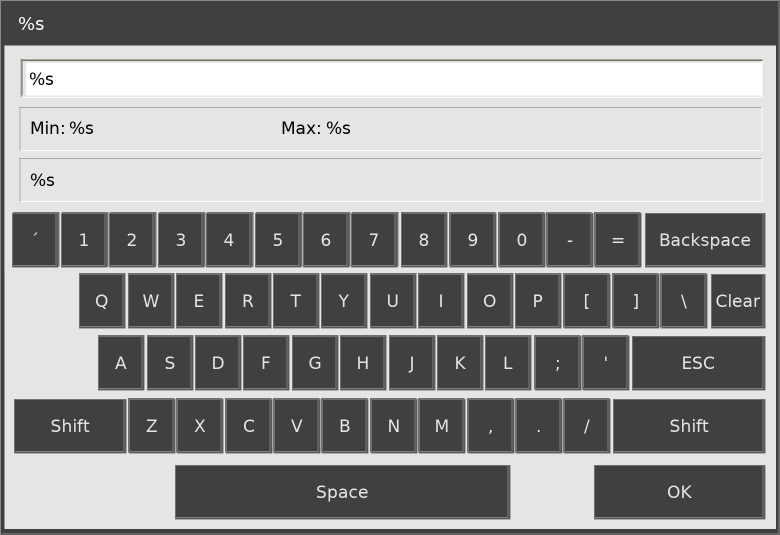
VISUALIZATION Keypad  // 780x535
VAR_INPUT
	stVariableValue 						: STRING;
	stMin 									: STRING;
	stMax 									: STRING;
	stTitle 								: STRING;
	flags 									: DWORD;
END_VAR
VAR
	bInit 									: BOOL;
	bShift 									: BOOL;
	stMessage 								: STRING;
	stOutputValue 							: STRING;
END_VAR
    Rectangle (5,201 772x70)
    Rectangle (3,271 775x62)
    Rectangle (3,333 775x63)
    Rectangle (3,396 775x62)
    Rectangle (3,455 775x75)
    Button (594,465 171x54), "OK"
        OnMouseDown: CloseDialog Dialog=Keypad, Result=OK, NumpadKeypad=True, NumpadKeypadSet=True
    Button (632,336 133x54), "ESC"
        OnMouseDown: CloseDialog Dialog=Keypad, Result=Cancel, NumpadKeypad=True, NumpadKeypadSet=True
    Button (711,274 54x54), "Clear"
        OnMouseDown: execute { stVariableValue := ''; stOutputValue := ''; }
    Button (645,213 120x54), "Backspace"
        OnMouseDown: execute { VisuDlg_CheckedBack(stOutputValue, stVariableValue, bInit); }
    Button (613,399 152x54), "Shift"
        OnMouseDown: toggle bShift
    Button (175,465 335x54), "Space"
        OnMouseDown: execute { VisuDlg_CheckedAppend(stOutputValue, stVariableValue, bInit, (flags AND VisuElems.Visu_InputFlags.Password) = 1, ' '); }
    Button (660,273 46x54), "|", invisible if: NOT bShift
        OnMouseDown: execute { VisuDlg_CheckedAppend(stOutputValue, stVariableValue, bInit, (flags AND VisuElems.Visu_InputFlags.Password) = 1, '|'); }
    Button (467,398 46x54), "<", invisible if: NOT bShift
        OnMouseDown: execute { VisuDlg_CheckedAppend(stOutputValue, stVariableValue, bInit, (flags AND VisuElems.Visu_InputFlags.Password) = 1, '<'); }
    Button (515,398 46x54), ">", invisible if: NOT bShift
        OnMouseDown: execute { VisuDlg_CheckedAppend(stOutputValue, stVariableValue, bInit, (flags AND VisuElems.Visu_InputFlags.Password) = 1, '>'); }
    Button (321,273 46x54), "y", invisible if: NOT bShift
        OnMouseDown: execute { VisuDlg_CheckedAppend(stOutputValue, stVariableValue, bInit, (flags AND VisuElems.Visu_InputFlags.Password) = 1, 'y'); }
    Button (321,274 46x54), "Y", invisible if: bShift
        OnMouseDown: execute { VisuDlg_CheckedAppend(stOutputValue, stVariableValue, bInit, (flags AND VisuElems.Visu_InputFlags.Password) = 1, 'Y'); }
    Button (176,398 46x54), "x", invisible if: NOT bShift
        OnMouseDown: execute { VisuDlg_CheckedAppend(stOutputValue, stVariableValue, bInit, (flags AND VisuElems.Visu_InputFlags.Password) = 1, 'x'); }
    Button (177,399 46x54), "X", invisible if: bShift
        OnMouseDown: execute { VisuDlg_CheckedAppend(stOutputValue, stVariableValue, bInit, (flags AND VisuElems.Visu_InputFlags.Password) = 1, 'X'); }
    Button (225,398 46x54), "c", invisible if: NOT bShift
        OnMouseDown: execute { VisuDlg_CheckedAppend(stOutputValue, stVariableValue, bInit, (flags AND VisuElems.Visu_InputFlags.Password) = 1, 'c'); }
    Button (226,399 46x54), "C", invisible if: bShift
        OnMouseDown: execute { VisuDlg_CheckedAppend(stOutputValue, stVariableValue, bInit, (flags AND VisuElems.Visu_InputFlags.Password) = 1, 'C'); }
    Button (273,398 46x54), "v", invisible if: NOT bShift
        OnMouseDown: execute { VisuDlg_CheckedAppend(stOutputValue, stVariableValue, bInit, (flags AND VisuElems.Visu_InputFlags.Password) = 1, 'v'); }
    Button (274,399 46x54), "V", invisible if: bShift
        OnMouseDown: execute { VisuDlg_CheckedAppend(stOutputValue, stVariableValue, bInit, (flags AND VisuElems.Visu_InputFlags.Password) = 1, 'V'); }
    Button (321,398 46x54), "b", invisible if: NOT bShift
        OnMouseDown: execute { VisuDlg_CheckedAppend(stOutputValue, stVariableValue, bInit, (flags AND VisuElems.Visu_InputFlags.Password) = 1, 'b'); }
    Button (322,399 46x54), "B", invisible if: bShift
        OnMouseDown: execute { VisuDlg_CheckedAppend(stOutputValue, stVariableValue, bInit, (flags AND VisuElems.Visu_InputFlags.Password) = 1, 'B'); }
    Button (370,398 46x54), "n", invisible if: NOT bShift
        OnMouseDown: execute { VisuDlg_CheckedAppend(stOutputValue, stVariableValue, bInit, (flags AND VisuElems.Visu_InputFlags.Password) = 1, 'n'); }
    Button (371,399 46x54), "N", invisible if: bShift
        OnMouseDown: execute { VisuDlg_CheckedAppend(stOutputValue, stVariableValue, bInit, (flags AND VisuElems.Visu_InputFlags.Password) = 1, 'N'); }
    Button (418,398 46x54), "m", invisible if: NOT bShift
        OnMouseDown: execute { VisuDlg_CheckedAppend(stOutputValue, stVariableValue, bInit, (flags AND VisuElems.Visu_InputFlags.Password) = 1, 'm'); }
    Button (419,399 46x54), "M", invisible if: bShift
        OnMouseDown: execute { VisuDlg_CheckedAppend(stOutputValue, stVariableValue, bInit, (flags AND VisuElems.Visu_InputFlags.Password) = 1, 'M'); }
    Button (534,335 46x54), ":", invisible if: NOT bShift
        OnMouseDown: execute { VisuDlg_CheckedAppend(stOutputValue, stVariableValue, bInit, (flags AND VisuElems.Visu_InputFlags.Password) = 1, ':'); }
    Button (546,212 45x54), "_", invisible if: NOT bShift
        OnMouseDown: execute { VisuDlg_CheckedAppend(stOutputValue, stVariableValue, bInit, (flags AND VisuElems.Visu_InputFlags.Password) = 1, '_'); }
    Button (98,335 46x54), "a", invisible if: NOT bShift
        OnMouseDown: execute { VisuDlg_CheckedAppend(stOutputValue, stVariableValue, bInit, (flags AND VisuElems.Visu_InputFlags.Password) = 1, 'a'); }
    Button (98,336 46x54), "A", invisible if: bShift
        OnMouseDown: execute { VisuDlg_CheckedAppend(stOutputValue, stVariableValue, bInit, (flags AND VisuElems.Visu_InputFlags.Password) = 1, 'A'); }
    Button (147,335 46x54), "s", invisible if: NOT bShift
        OnMouseDown: execute { VisuDlg_CheckedAppend(stOutputValue, stVariableValue, bInit, (flags AND VisuElems.Visu_InputFlags.Password) = 1, 's'); }
    Button (147,336 46x54), "S", invisible if: bShift
        OnMouseDown: execute { VisuDlg_CheckedAppend(stOutputValue, stVariableValue, bInit, (flags AND VisuElems.Visu_InputFlags.Password) = 1, 'S'); }
    Button (195,335 46x54), "d", invisible if: NOT bShift
        OnMouseDown: execute { VisuDlg_CheckedAppend(stOutputValue, stVariableValue, bInit, (flags AND VisuElems.Visu_InputFlags.Password) = 1, 'd'); }
    Button (195,336 46x54), "D", invisible if: bShift
        OnMouseDown: execute { VisuDlg_CheckedAppend(stOutputValue, stVariableValue, bInit, (flags AND VisuElems.Visu_InputFlags.Password) = 1, 'D'); }
    Button (243,335 46x54), "f", invisible if: NOT bShift
        OnMouseDown: execute { VisuDlg_CheckedAppend(stOutputValue, stVariableValue, bInit, (flags AND VisuElems.Visu_InputFlags.Password) = 1, 'f'); }
    Button (243,336 46x54), "F", invisible if: bShift
        OnMouseDown: execute { VisuDlg_CheckedAppend(stOutputValue, stVariableValue, bInit, (flags AND VisuElems.Visu_InputFlags.Password) = 1, 'F'); }
    Button (292,335 46x54), "g", invisible if: NOT bShift
        OnMouseDown: execute { VisuDlg_CheckedAppend(stOutputValue, stVariableValue, bInit, (flags AND VisuElems.Visu_InputFlags.Password) = 1, 'g'); }
    Button (292,336 46x54), "G", invisible if: bShift
        OnMouseDown: execute { VisuDlg_CheckedAppend(stOutputValue, stVariableValue, bInit, (flags AND VisuElems.Visu_InputFlags.Password) = 1, 'G'); }
    Button (340,335 46x54), "h", invisible if: NOT bShift
        OnMouseDown: execute { VisuDlg_CheckedAppend(stOutputValue, stVariableValue, bInit, (flags AND VisuElems.Visu_InputFlags.Password) = 1, 'h'); }
    Button (340,336 46x54), "H", invisible if: bShift
        OnMouseDown: execute { VisuDlg_CheckedAppend(stOutputValue, stVariableValue, bInit, (flags AND VisuElems.Visu_InputFlags.Password) = 1, 'H'); }
    Button (389,335 46x54), "j", invisible if: NOT bShift
        OnMouseDown: execute { VisuDlg_CheckedAppend(stOutputValue, stVariableValue, bInit, (flags AND VisuElems.Visu_InputFlags.Password) = 1, 'j'); }
    Button (389,336 46x54), "J", invisible if: bShift
        OnMouseDown: execute { VisuDlg_CheckedAppend(stOutputValue, stVariableValue, bInit, (flags AND VisuElems.Visu_InputFlags.Password) = 1, 'J'); }
    Button (437,335 46x54), "k", invisible if: NOT bShift
        OnMouseDown: execute { VisuDlg_CheckedAppend(stOutputValue, stVariableValue, bInit, (flags AND VisuElems.Visu_InputFlags.Password) = 1, 'k'); }
    Button (437,336 46x54), "K", invisible if: bShift
        OnMouseDown: execute { VisuDlg_CheckedAppend(stOutputValue, stVariableValue, bInit, (flags AND VisuElems.Visu_InputFlags.Password) = 1, 'K'); }
    Button (485,335 46x54), "l", invisible if: NOT bShift
        OnMouseDown: execute { VisuDlg_CheckedAppend(stOutputValue, stVariableValue, bInit, (flags AND VisuElems.Visu_InputFlags.Password) = 1, 'l'); }
    Button (485,336 46x54), "L", invisible if: bShift
        OnMouseDown: execute { VisuDlg_CheckedAppend(stOutputValue, stVariableValue, bInit, (flags AND VisuElems.Visu_InputFlags.Password) = 1, 'L'); }
    Button (159,212 46x54), "#", invisible if: NOT bShift
        OnMouseDown: execute { VisuDlg_CheckedAppend(stOutputValue, stVariableValue, bInit, (flags AND VisuElems.Visu_InputFlags.Password) = 1, '#'); }
    Button (110,212 46x54), "@", invisible if: NOT bShift
        OnMouseDown: execute { VisuDlg_CheckedAppend(stOutputValue, stVariableValue, bInit, (flags AND VisuElems.Visu_InputFlags.Password) = 1, '@'); }
    Button (79,273 46x54), "q", invisible if: NOT bShift
        OnMouseDown: execute { VisuDlg_CheckedAppend(stOutputValue, stVariableValue, bInit, (flags AND VisuElems.Visu_InputFlags.Password) = 1, 'q'); }
    Button (79,274 46x54), "Q", invisible if: bShift
        OnMouseDown: execute { VisuDlg_CheckedAppend(stOutputValue, stVariableValue, bInit, (flags AND VisuElems.Visu_InputFlags.Password) = 1, 'Q'); }
    Button (128,273 46x54), "w", invisible if: NOT bShift
        OnMouseDown: execute { VisuDlg_CheckedAppend(stOutputValue, stVariableValue, bInit, (flags AND VisuElems.Visu_InputFlags.Password) = 1, 'w'); }
    Button (128,274 46x54), "W", invisible if: bShift
        OnMouseDown: execute { VisuDlg_CheckedAppend(stOutputValue, stVariableValue, bInit, (flags AND VisuElems.Visu_InputFlags.Password) = 1, 'W'); }
    Button (176,273 46x54), "e", invisible if: NOT bShift
        OnMouseDown: execute { VisuDlg_CheckedAppend(stOutputValue, stVariableValue, bInit, (flags AND VisuElems.Visu_InputFlags.Password) = 1, 'e'); }
    Button (176,274 46x54), "E", invisible if: bShift
        OnMouseDown: execute { VisuDlg_CheckedAppend(stOutputValue, stVariableValue, bInit, (flags AND VisuElems.Visu_InputFlags.Password) = 1, 'E'); }
    Button (225,273 46x54), "r", invisible if: NOT bShift
        OnMouseDown: execute { VisuDlg_CheckedAppend(stOutputValue, stVariableValue, bInit, (flags AND VisuElems.Visu_InputFlags.Password) = 1, 'r'); }
    Button (225,274 46x54), "R", invisible if: bShift
        OnMouseDown: execute { VisuDlg_CheckedAppend(stOutputValue, stVariableValue, bInit, (flags AND VisuElems.Visu_InputFlags.Password) = 1, 'R'); }
    Button (273,273 46x54), "t", invisible if: NOT bShift
        OnMouseDown: execute { VisuDlg_CheckedAppend(stOutputValue, stVariableValue, bInit, (flags AND VisuElems.Visu_InputFlags.Password) = 1, 't'); }
    Button (273,274 46x54), "T", invisible if: bShift
        OnMouseDown: execute { VisuDlg_CheckedAppend(stOutputValue, stVariableValue, bInit, (flags AND VisuElems.Visu_InputFlags.Password) = 1, 'T'); }
    Button (128,398 46x54), "z", invisible if: NOT bShift
        OnMouseDown: execute { VisuDlg_CheckedAppend(stOutputValue, stVariableValue, bInit, (flags AND VisuElems.Visu_InputFlags.Password) = 1, 'z'); }
    Button (129,399 46x54), "Z", invisible if: bShift
        OnMouseDown: execute { VisuDlg_CheckedAppend(stOutputValue, stVariableValue, bInit, (flags AND VisuElems.Visu_InputFlags.Password) = 1, 'Z'); }
    Button (370,273 46x54), "u", invisible if: NOT bShift
        OnMouseDown: execute { VisuDlg_CheckedAppend(stOutputValue, stVariableValue, bInit, (flags AND VisuElems.Visu_InputFlags.Password) = 1, 'u'); }
    Button (370,274 46x54), "U", invisible if: bShift
        OnMouseDown: execute { VisuDlg_CheckedAppend(stOutputValue, stVariableValue, bInit, (flags AND VisuElems.Visu_InputFlags.Password) = 1, 'U'); }
    Button (418,273 46x54), "i", invisible if: NOT bShift
        OnMouseDown: execute { VisuDlg_CheckedAppend(stOutputValue, stVariableValue, bInit, (flags AND VisuElems.Visu_InputFlags.Password) = 1, 'i'); }
    Button (418,274 46x54), "I", invisible if: bShift
        OnMouseDown: execute { VisuDlg_CheckedAppend(stOutputValue, stVariableValue, bInit, (flags AND VisuElems.Visu_InputFlags.Password) = 1, 'I'); }
    Button (467,273 46x54), "o", invisible if: NOT bShift
        OnMouseDown: execute { VisuDlg_CheckedAppend(stOutputValue, stVariableValue, bInit, (flags AND VisuElems.Visu_InputFlags.Password) = 1, 'o'); }
    Button (467,274 46x54), "O", invisible if: bShift
        OnMouseDown: execute { VisuDlg_CheckedAppend(stOutputValue, stVariableValue, bInit, (flags AND VisuElems.Visu_InputFlags.Password) = 1, 'O'); }
    Button (515,273 46x54), "p", invisible if: NOT bShift
        OnMouseDown: execute { VisuDlg_CheckedAppend(stOutputValue, stVariableValue, bInit, (flags AND VisuElems.Visu_InputFlags.Password) = 1, 'p'); }
    Button (515,274 46x54), "P", invisible if: bShift
        OnMouseDown: execute { VisuDlg_CheckedAppend(stOutputValue, stVariableValue, bInit, (flags AND VisuElems.Visu_InputFlags.Password) = 1, 'P'); }
    Button (594,212 46x54), "+", invisible if: NOT bShift
        OnMouseDown: execute { VisuDlg_CheckedAppend(stOutputValue, stVariableValue, bInit, (flags AND VisuElems.Visu_InputFlags.Password) = 1, '+'); }
    Button (401,212 46x54), "*", invisible if: NOT bShift
        OnMouseDown: execute { VisuDlg_CheckedAppend(stOutputValue, stVariableValue, bInit, (flags AND VisuElems.Visu_InputFlags.Password) = 1, '*'); }
    Button (13,212 46x54), "~", invisible if: NOT bShift
        OnMouseDown: execute { VisuDlg_CheckedAppend(stOutputValue, stVariableValue, bInit, (flags AND VisuElems.Visu_InputFlags.Password) = 1, '~'); }
    Button (304,212 46x54), "^", invisible if: NOT bShift
        OnMouseDown: execute { VisuDlg_CheckedAppend(stOutputValue, stVariableValue, bInit, (flags AND VisuElems.Visu_InputFlags.Password) = 1, '^'); }
    Button (62,212 46x54), "!", invisible if: NOT bShift
        OnMouseDown: execute { VisuDlg_CheckedAppend(stOutputValue, stVariableValue, bInit, (flags AND VisuElems.Visu_InputFlags.Password) = 1, '!'); }
    Button (582,335 46x54), """, invisible if: NOT bShift
        OnMouseDown: execute { VisuDlg_CheckedAppend(stOutputValue, stVariableValue, bInit, (flags AND VisuElems.Visu_InputFlags.Password) = 1, '"'); }
    Button (207,212 46x54), "$", invisible if: NOT bShift
        OnMouseDown: execute { VisuDlg_CheckedAppend(stOutputValue, stVariableValue, bInit, (flags AND VisuElems.Visu_InputFlags.Password) = 1, '$$'); }
    Button (256,212 46x54), "%", invisible if: NOT bShift
        OnMouseDown: execute { VisuDlg_CheckedAppend(stOutputValue, stVariableValue, bInit, (flags AND VisuElems.Visu_InputFlags.Password) = 1, '%'); }
    Button (352,212 46x54), "&", invisible if: NOT bShift
        OnMouseDown: execute { VisuDlg_CheckedAppend(stOutputValue, stVariableValue, bInit, (flags AND VisuElems.Visu_InputFlags.Password) = 1, '&'); }
    Button (449,212 46x54), "(", invisible if: NOT bShift
        OnMouseDown: execute { VisuDlg_CheckedAppend(stOutputValue, stVariableValue, bInit, (flags AND VisuElems.Visu_InputFlags.Password) = 1, '('); }
    Button (498,212 46x54), ")", invisible if: NOT bShift
        OnMouseDown: execute { VisuDlg_CheckedAppend(stOutputValue, stVariableValue, bInit, (flags AND VisuElems.Visu_InputFlags.Password) = 1, ')'); }
    Button (563,398 46x54), "?", invisible if: NOT bShift
        OnMouseDown: execute { VisuDlg_CheckedAppend(stOutputValue, stVariableValue, bInit, (flags AND VisuElems.Visu_InputFlags.Password) = 1, '?'); }
    Rectangle (5,104 773x97)
    Rectangle (27,164 734x32), "%s", text variable: stMessage
    Rectangle (5,42 773x62)
    Rectangle (776,0 4x530)
    Rectangle (0,2 4x527)
    Rectangle (0,529 780x6)
    Polyline (20,201) (20,158) (762,158)
    Polyline (20,150) (20,107) (762,107)
    Polyline (21,97) (21,59) (762,59)
    Polyline (21,201) (762,201) (762,158)
    Polyline (21,150) (762,150) (762,107)
    Polyline (22,97) (762,97) (762,60)
    Rectangle (0,0 779x45)
    Rectangle (15,8 757x32), "%s", text variable: stTitle
    Polyline (22,95) (22,60) (762,60)
    Rectangle (26,63 736x32), "%s", text variable: stOutputValue
    Rectangle (27,112 42x32), "Min:", text variable: stMin, invisible if: LEN(stMin) = 0
    Rectangle (66,112 157x32), "%s", text variable: stMin, invisible if: LEN(stMin) = 0
    Rectangle (278,112 45x32), "Max:", text variable: stMin, invisible if: LEN(stMax) = 0
    Rectangle (323,112 217x32), "%s", text variable: stMax, invisible if: LEN(stMax) = 0
    Button (12,213 46x54), "´", invisible if: bShift
        OnMouseDown: execute { VisuDlg_CheckedAppend(stOutputValue, stVariableValue, bInit, (flags AND VisuElems.Visu_InputFlags.Password) = 1, '´'); }
    Button (61,213 46x54), "1", invisible if: bShift
        OnMouseDown: execute { VisuDlg_CheckedAppend(stOutputValue, stVariableValue, bInit, (flags AND VisuElems.Visu_InputFlags.Password) = 1, '1'); }
    Button (109,213 46x54), "2", invisible if: bShift
        OnMouseDown: execute { VisuDlg_CheckedAppend(stOutputValue, stVariableValue, bInit, (flags AND VisuElems.Visu_InputFlags.Password) = 1, '2'); }
    Button (158,213 46x54), "3", invisible if: bShift
        OnMouseDown: execute { VisuDlg_CheckedAppend(stOutputValue, stVariableValue, bInit, (flags AND VisuElems.Visu_InputFlags.Password) = 1, '3'); }
    Button (206,213 46x54), "4", invisible if: bShift
        OnMouseDown: execute { VisuDlg_CheckedAppend(stOutputValue, stVariableValue, bInit, (flags AND VisuElems.Visu_InputFlags.Password) = 1, '4'); }
    Button (255,213 46x54), "5", invisible if: bShift
        OnMouseDown: execute { VisuDlg_CheckedAppend(stOutputValue, stVariableValue, bInit, (flags AND VisuElems.Visu_InputFlags.Password) = 1, '5'); }
    Button (303,213 46x54), "6", invisible if: bShift
        OnMouseDown: execute { VisuDlg_CheckedAppend(stOutputValue, stVariableValue, bInit, (flags AND VisuElems.Visu_InputFlags.Password) = 1, '6'); }
    Button (351,213 46x54), "7", invisible if: bShift
        OnMouseDown: execute { VisuDlg_CheckedAppend(stOutputValue, stVariableValue, bInit, (flags AND VisuElems.Visu_InputFlags.Password) = 1, '7'); }
    Button (401,213 46x54), "8", invisible if: bShift
        OnMouseDown: execute { VisuDlg_CheckedAppend(stOutputValue, stVariableValue, bInit, (flags AND VisuElems.Visu_InputFlags.Password) = 1, '8'); }
    Button (450,213 46x54), "9", invisible if: bShift
        OnMouseDown: execute { VisuDlg_CheckedAppend(stOutputValue, stVariableValue, bInit, (flags AND VisuElems.Visu_InputFlags.Password) = 1, '9'); }
    Button (499,213 46x54), "0", invisible if: bShift
        OnMouseDown: execute { VisuDlg_CheckedAppend(stOutputValue, stVariableValue, bInit, (flags AND VisuElems.Visu_InputFlags.Password) = 1, '0'); }
    Button (547,213 46x54), "-", invisible if: bShift
        OnMouseDown: execute { VisuDlg_CheckedAppend(stOutputValue, stVariableValue, bInit, (flags AND VisuElems.Visu_InputFlags.Password) = 1, '-'); }
    Button (595,213 46x54), "=", invisible if: bShift
        OnMouseDown: execute { VisuDlg_CheckedAppend(stOutputValue, stVariableValue, bInit, (flags AND VisuElems.Visu_InputFlags.Password) = 1, '='); }
    Button (563,273 46x54), "{", invisible if: NOT bShift
        OnMouseDown: execute { VisuDlg_CheckedAppend(stOutputValue, stVariableValue, bInit, (flags AND VisuElems.Visu_InputFlags.Password) = 1, '{'); }
    Button (564,274 46x54), "[", invisible if: bShift
        OnMouseDown: execute { VisuDlg_CheckedAppend(stOutputValue, stVariableValue, bInit, (flags AND VisuElems.Visu_InputFlags.Password) = 1, '['); }
    Button (612,273 46x54), "}", invisible if: NOT bShift
        OnMouseDown: execute { VisuDlg_CheckedAppend(stOutputValue, stVariableValue, bInit, (flags AND VisuElems.Visu_InputFlags.Password) = 1, '}'); }
    Button (613,274 46x54), "]", invisible if: bShift
        OnMouseDown: execute { VisuDlg_CheckedAppend(stOutputValue, stVariableValue, bInit, (flags AND VisuElems.Visu_InputFlags.Password) = 1, ']'); }
    Button (661,274 46x54), "\", invisible if: bShift
        OnMouseDown: execute { VisuDlg_CheckedAppend(stOutputValue, stVariableValue, bInit, (flags AND VisuElems.Visu_InputFlags.Password) = 1, '\'); }
    Button (535,336 46x54), ";", invisible if: bShift
        OnMouseDown: execute { VisuDlg_CheckedAppend(stOutputValue, stVariableValue, bInit, (flags AND VisuElems.Visu_InputFlags.Password) = 1, ';'); }
    Button (583,336 46x54), "'", invisible if: bShift
        OnMouseDown: execute { VisuDlg_CheckedAppend(stOutputValue, stVariableValue, bInit, (flags AND VisuElems.Visu_InputFlags.Password) = 1, '$''); }
    Button (468,399 46x54), ",", invisible if: bShift
        OnMouseDown: execute { VisuDlg_CheckedAppend(stOutputValue, stVariableValue, bInit, (flags AND VisuElems.Visu_InputFlags.Password) = 1, ','); }
    Button (516,399 46x54), ".", invisible if: bShift
        OnMouseDown: execute { VisuDlg_CheckedAppend(stOutputValue, stVariableValue, bInit, (flags AND VisuElems.Visu_InputFlags.Password) = 1, '.'); }
    Button (564,399 46x54), "/", invisible if: bShift
        OnMouseDown: execute { VisuDlg_CheckedAppend(stOutputValue, stVariableValue, bInit, (flags AND VisuElems.Visu_InputFlags.Password) = 1, '/'); }
    Button (14,399 112x54), "Shift"
        OnMouseDown: toggle bShift
    hotkey HotkeyInput Id=481083523072, Key=KeyDown=True, KeyName=BACKSPACE, ActionToExecute=Action=STSnippet=VisuDlg_CheckedBack(stOutputValue, stVariableValue, bInit);, VisuElemId=-1
    hotkey HotkeyInput Id=481084571648, Key=KeyDown=True, KeyName=DELETE, ActionToExecute=Action=STSnippet=stVariableValue := ''; stOutputValue := '';, VisuElemId=-1
    hotkey HotkeyInput Id=481085620224, Key=KeyDown=True, KeyName=ESCAPE, ActionToExecute=Action=Dialog=Keypad, Result=Cancel, NumpadKeypad=True, NumpadKeypadSet=True, VisuElemId=-1
    hotkey HotkeyInput Id=481086668800, Key=KeyDown=True, KeyName=SPACE, ActionToExecute=Action=STSnippet=VisuDlg_CheckedAppend(stOutputValue, stVariableValue, bInit, (flags AND VisuElems.Visu_InputFlags.Password) = 1, ' ');, VisuElemId=-1
    hotkey HotkeyInput Id=481087717376, Key=Modifiers=1, KeyDown=True, KeyName=SPACE, ActionToExecute=Action=ToggleVariable=bShift, VisuElemId=-1
    hotkey HotkeyInput Id=481088765952, Key=KeyDown=True, KeyName=RETURN_KEY, ActionToExecute=Action=Dialog=Keypad, Result=OK, NumpadKeypad=True, NumpadKeypadSet=True, VisuElemId=-1
    hotkey HotkeyInput Id=481089814528, Key=KeyDown=True, KeyName=1, ActionToExecute=Action=STSnippet=IF bShift THEN VisuDlg_CheckedAppend(stOutputValue, stVariableValue, bInit, (flags AND VisuElems.Visu_InputFlags.Password) = 1, '!'); ELSE VisuDlg_CheckedAppend(stOutputValue, stVariableValue, bInit, (flags AND VisuElems.Visu_InputFlags.Password) = 1, '1'); END_IF, VisuElemId=-1
    hotkey HotkeyInput Id=481090863104, Key=KeyDown=True, KeyName=2, ActionToExecute=Action=STSnippet=IF bShift THEN VisuDlg_CheckedAppend(stOutputValue, stVariableValue, bInit, (flags AND VisuElems.Visu_InputFlags.Password) = 1, '@'); ELSE VisuDlg_CheckedAppend(stOutputValue, stVariableValue, bInit, (flags AND VisuElems.Visu_InputFlags.Password) = 1, '2'); END_IF, VisuElemId=-1
    hotkey HotkeyInput Id=481091911680, Key=KeyDown=True, KeyName=3, ActionToExecute=Action=STSnippet=IF bShift THEN VisuDlg_CheckedAppend(stOutputValue, stVariableValue, bInit, (flags AND VisuElems.Visu_InputFlags.Password) = 1, '#'); ELSE VisuDlg_CheckedAppend(stOutputValue, stVariableValue, bInit, (flags AND VisuElems.Visu_InputFlags.Password) = 1, '3'); END_IF, VisuElemId=-1
    hotkey HotkeyInput Id=481092960256, Key=KeyDown=True, KeyName=4, ActionToExecute=Action=STSnippet=IF bShift THEN VisuDlg_CheckedAppend(stOutputValue, stVariableValue, bInit, (flags AND VisuElems.Visu_InputFlags.Password) = 1, '$$'); ELSE VisuDlg_CheckedAppend(stOutputValue, stVariableValue, bInit, (flags AND VisuElems.Visu_InputFlags.Password) = 1, '4'); END_IF, VisuElemId=-1
    hotkey HotkeyInput Id=481094008832, Key=KeyDown=True, KeyName=5, ActionToExecute=Action=STSnippet=IF bShift THEN VisuDlg_CheckedAppend(stOutputValue, stVariableValue, bInit, (flags AND VisuElems.Visu_InputFlags.Password) = 1, '%'); ELSE VisuDlg_CheckedAppend(stOutputValue, stVariableValue, bInit, (flags AND VisuElems.Visu_InputFlags.Password) = 1, '5'); END_IF, VisuElemId=-1
    hotkey HotkeyInput Id=481095057408, Key=KeyDown=True, KeyName=6, ActionToExecute=Action=STSnippet=IF bShift THEN VisuDlg_CheckedAppend(stOutputValue, stVariableValue, bInit, (flags AND VisuElems.Visu_InputFlags.Password) = 1, '^'); ELSE VisuDlg_CheckedAppend(stOutputValue, stVariableValue, bInit, (flags AND VisuElems.Visu_InputFlags.Password) = 1, '6'); END_IF, VisuElemId=-1
    hotkey HotkeyInput Id=481096105984, Key=KeyDown=True, KeyName=7, ActionToExecute=Action=STSnippet=IF bShift THEN VisuDlg_CheckedAppend(stOutputValue, stVariableValue, bInit, (flags AND VisuElems.Visu_InputFlags.Password) = 1, '&'); ELSE VisuDlg_CheckedAppend(stOutputValue, stVariableValue, bInit, (flags AND VisuElems.Visu_InputFlags.Password) = 1, '7'); END_IF, VisuElemId=-1
    hotkey HotkeyInput Id=481097154560, Key=KeyDown=True, KeyName=8, ActionToExecute=Action=STSnippet=IF bShift THEN VisuDlg_CheckedAppend(stOutputValue, stVariableValue, bInit, (flags AND VisuElems.Visu_InputFlags.Password) = 1, '*'); ELSE VisuDlg_CheckedAppend(stOutputValue, stVariableValue, bInit, (flags AND VisuElems.Visu_InputFlags.Password) = 1, '8'); END_IF, VisuElemId=-1
    hotkey HotkeyInput Id=481098203136, Key=KeyDown=True, KeyName=9, ActionToExecute=Action=STSnippet=IF bShift THEN VisuDlg_CheckedAppend(stOutputValue, stVariableValue, bInit, (flags AND VisuElems.Visu_InputFlags.Password) = 1, '('); ELSE VisuDlg_CheckedAppend(stOutputValue, stVariableValue, bInit, (flags AND VisuElems.Visu_InputFlags.Password) = 1, '9'); END_IF, VisuElemId=-1
    hotkey HotkeyInput Id=481099251712, Key=KeyDown=True, KeyName=0, ActionToExecute=Action=STSnippet=IF bShift THEN VisuDlg_CheckedAppend(stOutputValue, stVariableValue, bInit, (flags AND VisuElems.Visu_InputFlags.Password) = 1, ')'); ELSE VisuDlg_CheckedAppend(stOutputValue, stVariableValue, bInit, (flags AND VisuElems.Visu_InputFlags.Password) = 1, '0'); END_IF, VisuElemId=-1
    hotkey HotkeyInput Id=481100300288, Key=KeyDown=True, KeyName=SUBTRACT, ActionToExecute=Action=STSnippet=IF bShift THEN VisuDlg_CheckedAppend(stOutputValue, stVariableValue, bInit, (flags AND VisuElems.Visu_InputFlags.Password) = 1, '_'); ELSE VisuDlg_CheckedAppend(stOutputValue, stVariableValue, bInit, (flags AND VisuElems.Visu_InputFlags.Password) = 1, '-'); END_IF, VisuElemId=-1
    hotkey HotkeyInput Id=481101348864, Key=KeyDown=True, KeyName=ADDITION, ActionToExecute=Action=STSnippet=IF bShift THEN VisuDlg_CheckedAppend(stOutputValue, stVariableValue, bInit, (flags AND VisuElems.Visu_InputFlags.Password) = 1, '='); ELSE VisuDlg_CheckedAppend(stOutputValue, stVariableValue, bInit, (flags AND VisuElems.Visu_InputFlags.Password) = 1, '+'); END_IF, VisuElemId=-1
    hotkey HotkeyInput Id=481102397440, Key=KeyDown=True, KeyName=Q, ActionToExecute=Action=STSnippet=IF bShift THEN VisuDlg_CheckedAppend(stOutputValue, stVariableValue, bInit, (flags AND VisuElems.Visu_InputFlags.Password) = 1, 'q'); ELSE VisuDlg_CheckedAppend(stOutputValue, stVariableValue, bInit, (flags AND VisuElems.Visu_InputFlags.Password) = 1, 'Q'); END_IF, VisuElemId=-1
    hotkey HotkeyInput Id=481103446016, Key=KeyDown=True, KeyName=W, ActionToExecute=Action=STSnippet=IF bShift THEN VisuDlg_CheckedAppend(stOutputValue, stVariableValue, bInit, (flags AND VisuElems.Visu_InputFlags.Password) = 1, 'w'); ELSE VisuDlg_CheckedAppend(stOutputValue, stVariableValue, bInit, (flags AND VisuElems.Visu_InputFlags.Password) = 1, 'W'); END_IF, VisuElemId=-1
    hotkey HotkeyInput Id=481104494592, Key=KeyDown=True, KeyName=E, ActionToExecute=Action=STSnippet=IF bShift THEN VisuDlg_CheckedAppend(stOutputValue, stVariableValue, bInit, (flags AND VisuElems.Visu_InputFlags.Password) = 1, 'e'); ELSE VisuDlg_CheckedAppend(stOutputValue, stVariableValue, bInit, (flags AND VisuElems.Visu_InputFlags.Password) = 1, 'E'); END_IF, VisuElemId=-1
    hotkey HotkeyInput Id=481105543168, Key=KeyDown=True, KeyName=R, ActionToExecute=Action=STSnippet=IF bShift THEN VisuDlg_CheckedAppend(stOutputValue, stVariableValue, bInit, (flags AND VisuElems.Visu_InputFlags.Password) = 1, 'r'); ELSE VisuDlg_CheckedAppend(stOutputValue, stVariableValue, bInit, (flags AND VisuElems.Visu_InputFlags.Password) = 1, 'R'); END_IF, VisuElemId=-1
    hotkey HotkeyInput Id=481106591744, Key=KeyDown=True, KeyName=T, ActionToExecute=Action=STSnippet=IF bShift THEN VisuDlg_CheckedAppend(stOutputValue, stVariableValue, bInit, (flags AND VisuElems.Visu_InputFlags.Password) = 1, 't'); ELSE VisuDlg_CheckedAppend(stOutputValue, stVariableValue, bInit, (flags AND VisuElems.Visu_InputFlags.Password) = 1, 'T'); END_IF, VisuElemId=-1
    hotkey HotkeyInput Id=481107640320, Key=KeyDown=True, KeyName=Y, ActionToExecute=Action=STSnippet=IF bShift THEN VisuDlg_CheckedAppend(stOutputValue, stVariableValue, bInit, (flags AND VisuElems.Visu_InputFlags.Password) = 1, 'y'); ELSE VisuDlg_CheckedAppend(stOutputValue, stVariableValue, bInit, (flags AND VisuElems.Visu_InputFlags.Password) = 1, 'Y'); END_IF, VisuElemId=-1
    hotkey HotkeyInput Id=481108688896, Key=KeyDown=True, KeyName=U, ActionToExecute=Action=STSnippet=IF bShift THEN VisuDlg_CheckedAppend(stOutputValue, stVariableValue, bInit, (flags AND VisuElems.Visu_InputFlags.Password) = 1, 'u'); ELSE VisuDlg_CheckedAppend(stOutputValue, stVariableValue, bInit, (flags AND VisuElems.Visu_InputFlags.Password) = 1, 'U'); END_IF, VisuElemId=-1
    hotkey HotkeyInput Id=481109737472, Key=KeyDown=True, KeyName=I, ActionToExecute=Action=STSnippet=IF bShift THEN VisuDlg_CheckedAppend(stOutputValue, stVariableValue, bInit, (flags AND VisuElems.Visu_InputFlags.Password) = 1, 'i'); ELSE VisuDlg_CheckedAppend(stOutputValue, stVariableValue, bInit, (flags AND VisuElems.Visu_InputFlags.Password) = 1, 'I'); END_IF, VisuElemId=-1
    hotkey HotkeyInput Id=481110786048, Key=KeyDown=True, KeyName=O, ActionToExecute=Action=STSnippet=IF bShift THEN VisuDlg_CheckedAppend(stOutputValue, stVariableValue, bInit, (flags AND VisuElems.Visu_InputFlags.Password) = 1, 'o'); ELSE VisuDlg_CheckedAppend(stOutputValue, stVariableValue, bInit, (flags AND VisuElems.Visu_InputFlags.Password) = 1, 'O'); END_IF, VisuElemId=-1
    hotkey HotkeyInput Id=481111834624, Key=KeyDown=True, KeyName=P, ActionToExecute=Action=STSnippet=IF bShift THEN VisuDlg_CheckedAppend(stOutputValue, stVariableValue, bInit, (flags AND VisuElems.Visu_InputFlags.Password) = 1, 'p'); ELSE VisuDlg_CheckedAppend(stOutputValue, stVariableValue, bInit, (flags AND VisuElems.Visu_InputFlags.Password) = 1, 'P'); END_IF, VisuElemId=-1
    hotkey HotkeyInput Id=481112883200, Key=KeyDown=True, KeyName=A, ActionToExecute=Action=STSnippet=IF bShift THEN VisuDlg_CheckedAppend(stOutputValue, stVariableValue, bInit, (flags AND VisuElems.Visu_InputFlags.Password) = 1, 'a'); ELSE VisuDlg_CheckedAppend(stOutputValue, stVariableValue, bInit, (flags AND VisuElems.Visu_InputFlags.Password) = 1, 'A'); END_IF, VisuElemId=-1
    hotkey HotkeyInput Id=481113931776, Key=KeyDown=True, KeyName=S, ActionToExecute=Action=STSnippet=IF bShift THEN VisuDlg_CheckedAppend(stOutputValue, stVariableValue, bInit, (flags AND VisuElems.Visu_InputFlags.Password) = 1, 's'); ELSE VisuDlg_CheckedAppend(stOutputValue, stVariableValue, bInit, (flags AND VisuElems.Visu_InputFlags.Password) = 1, 'S'); END_IF, VisuElemId=-1
    hotkey HotkeyInput Id=481114980352, Key=KeyDown=True, KeyName=D, ActionToExecute=Action=STSnippet=IF bShift THEN VisuDlg_CheckedAppend(stOutputValue, stVariableValue, bInit, (flags AND VisuElems.Visu_InputFlags.Password) = 1, 'd'); ELSE VisuDlg_CheckedAppend(stOutputValue, stVariableValue, bInit, (flags AND VisuElems.Visu_InputFlags.Password) = 1, 'D'); END_IF, VisuElemId=-1
    hotkey HotkeyInput Id=481116028928, Key=KeyDown=True, KeyName=F, ActionToExecute=Action=STSnippet=IF bShift THEN VisuDlg_CheckedAppend(stOutputValue, stVariableValue, bInit, (flags AND VisuElems.Visu_InputFlags.Password) = 1, 'f'); ELSE VisuDlg_CheckedAppend(stOutputValue, stVariableValue, bInit, (flags AND VisuElems.Visu_InputFlags.Password) = 1, 'F'); END_IF, VisuElemId=-1
    hotkey HotkeyInput Id=481117077504, Key=KeyDown=True, KeyName=G, ActionToExecute=Action=STSnippet=IF bShift THEN VisuDlg_CheckedAppend(stOutputValue, stVariableValue, bInit, (flags AND VisuElems.Visu_InputFlags.Password) = 1, 'g'); ELSE VisuDlg_CheckedAppend(stOutputValue, stVariableValue, bInit, (flags AND VisuElems.Visu_InputFlags.Password) = 1, 'G'); END_IF, VisuElemId=-1
    hotkey HotkeyInput Id=481118126080, Key=KeyDown=True, KeyName=H, ActionToExecute=Action=STSnippet=IF bShift THEN VisuDlg_CheckedAppend(stOutputValue, stVariableValue, bInit, (flags AND VisuElems.Visu_InputFlags.Password) = 1, 'h'); ELSE VisuDlg_CheckedAppend(stOutputValue, stVariableValue, bInit, (flags AND VisuElems.Visu_InputFlags.Password) = 1, 'H'); END_IF, VisuElemId=-1
    hotkey HotkeyInput Id=481119174656, Key=KeyDown=True, KeyName=J, ActionToExecute=Action=STSnippet=IF bShift THEN VisuDlg_CheckedAppend(stOutputValue, stVariableValue, bInit, (flags AND VisuElems.Visu_InputFlags.Password) = 1, 'j'); ELSE VisuDlg_CheckedAppend(stOutputValue, stVariableValue, bInit, (flags AND VisuElems.Visu_InputFlags.Password) = 1, 'J'); END_IF, VisuElemId=-1
    hotkey HotkeyInput Id=481120223232, Key=KeyDown=True, KeyName=K, ActionToExecute=Action=STSnippet=IF bShift THEN VisuDlg_CheckedAppend(stOutputValue, stVariableValue, bInit, (flags AND VisuElems.Visu_InputFlags.Password) = 1, 'k'); ELSE VisuDlg_CheckedAppend(stOutputValue, stVariableValue, bInit, (flags AND VisuElems.Visu_InputFlags.Password) = 1, 'K'); END_IF, VisuElemId=-1
    hotkey HotkeyInput Id=481121271808, Key=KeyDown=True, KeyName=L, ActionToExecute=Action=STSnippet=IF bShift THEN VisuDlg_CheckedAppend(stOutputValue, stVariableValue, bInit, (flags AND VisuElems.Visu_InputFlags.Password) = 1, 'l'); ELSE VisuDlg_CheckedAppend(stOutputValue, stVariableValue, bInit, (flags AND VisuElems.Visu_InputFlags.Password) = 1, 'L'); END_IF, VisuElemId=-1
    hotkey HotkeyInput Id=481122320384, Key=KeyDown=True, KeyName=Z, ActionToExecute=Action=STSnippet=IF bShift THEN VisuDlg_CheckedAppend(stOutputValue, stVariableValue, bInit, (flags AND VisuElems.Visu_InputFlags.Password) = 1, 'z'); ELSE VisuDlg_CheckedAppend(stOutputValue, stVariableValue, bInit, (flags AND VisuElems.Visu_InputFlags.Password) = 1, 'Z'); END_IF, VisuElemId=-1
    hotkey HotkeyInput Id=481123368960, Key=KeyDown=True, KeyName=X, ActionToExecute=Action=STSnippet=IF bShift THEN VisuDlg_CheckedAppend(stOutputValue, stVariableValue, bInit, (flags AND VisuElems.Visu_InputFlags.Password) = 1, 'x'); ELSE VisuDlg_CheckedAppend(stOutputValue, stVariableValue, bInit, (flags AND VisuElems.Visu_InputFlags.Password) = 1, 'X'); END_IF, VisuElemId=-1
    hotkey HotkeyInput Id=481124417536, Key=KeyDown=True, KeyName=C, ActionToExecute=Action=STSnippet=IF bShift THEN VisuDlg_CheckedAppend(stOutputValue, stVariableValue, bInit, (flags AND VisuElems.Visu_InputFlags.Password) = 1, 'c'); ELSE VisuDlg_CheckedAppend(stOutputValue, stVariableValue, bInit, (flags AND VisuElems.Visu_InputFlags.Password) = 1, 'C'); END_IF, VisuElemId=-1
    hotkey HotkeyInput Id=481125466112, Key=KeyDown=True, KeyName=V, ActionToExecute=Action=STSnippet=IF bShift THEN VisuDlg_CheckedAppend(stOutputValue, stVariableValue, bInit, (flags AND VisuElems.Visu_InputFlags.Password) = 1, 'v'); ELSE VisuDlg_CheckedAppend(stOutputValue, stVariableValue, bInit, (flags AND VisuElems.Visu_InputFlags.Password) = 1, 'V'); END_IF, VisuElemId=-1
    hotkey HotkeyInput Id=481126514688, Key=KeyDown=True, KeyName=B, ActionToExecute=Action=STSnippet=IF bShift THEN VisuDlg_CheckedAppend(stOutputValue, stVariableValue, bInit, (flags AND VisuElems.Visu_InputFlags.Password) = 1, 'b'); ELSE VisuDlg_CheckedAppend(stOutputValue, stVariableValue, bInit, (flags AND VisuElems.Visu_InputFlags.Password) = 1, 'B'); END_IF, VisuElemId=-1
    hotkey HotkeyInput Id=481127563264, Key=KeyDown=True, KeyName=N, ActionToExecute=Action=STSnippet=IF bShift THEN VisuDlg_CheckedAppend(stOutputValue, stVariableValue, bInit, (flags AND VisuElems.Visu_InputFlags.Password) = 1, 'n'); ELSE VisuDlg_CheckedAppend(stOutputValue, stVariableValue, bInit, (flags AND VisuElems.Visu_InputFlags.Password) = 1, 'N'); END_IF, VisuElemId=-1
    hotkey HotkeyInput Id=481128611840, Key=KeyDown=True, KeyName=M, ActionToExecute=Action=STSnippet=IF bShift THEN VisuDlg_CheckedAppend(stOutputValue, stVariableValue, bInit, (flags AND VisuElems.Visu_InputFlags.Password) = 1, 'm'); ELSE VisuDlg_CheckedAppend(stOutputValue, stVariableValue, bInit, (flags AND VisuElems.Visu_InputFlags.Password) = 1, 'M'); END_IF, VisuElemId=-1
    hotkey HotkeyInput Id=481129660416, Key=KeyDown=True, KeyName=COMMA, ActionToExecute=Action=STSnippet=IF bShift THEN VisuDlg_CheckedAppend(stOutputValue, stVariableValue, bInit, (flags AND VisuElems.Visu_InputFlags.Password) = 1, ','); ELSE VisuDlg_CheckedAppend(stOutputValue, stVariableValue, bInit, (flags AND VisuElems.Visu_InputFlags.Password) = 1, '.'); END_IF, VisuElemId=-1
    hotkey HotkeyInput Id=481131757568, Key=KeyDown=True, KeyName=NUM1, ActionToExecute=Action=STSnippet=VisuDlg_CheckedAppend(stOutputValue, stVariableValue, bInit, (flags AND VisuElems.Visu_InputFlags.Password) = 1, '1');, VisuElemId=-1
    hotkey HotkeyInput Id=481132806144, Key=KeyDown=True, KeyName=NUM2, ActionToExecute=Action=STSnippet=VisuDlg_CheckedAppend(stOutputValue, stVariableValue, bInit, (flags AND VisuElems.Visu_InputFlags.Password) = 1, '2');, VisuElemId=-1
    hotkey HotkeyInput Id=481133854720, Key=KeyDown=True, KeyName=NUM3, ActionToExecute=Action=STSnippet=VisuDlg_CheckedAppend(stOutputValue, stVariableValue, bInit, (flags AND VisuElems.Visu_InputFlags.Password) = 1, '3');, VisuElemId=-1
    hotkey HotkeyInput Id=481134903296, Key=KeyDown=True, KeyName=NUM4, ActionToExecute=Action=STSnippet=VisuDlg_CheckedAppend(stOutputValue, stVariableValue, bInit, (flags AND VisuElems.Visu_InputFlags.Password) = 1, '4');, VisuElemId=-1
    hotkey HotkeyInput Id=481135951872, Key=KeyDown=True, KeyName=NUM5, ActionToExecute=Action=STSnippet=VisuDlg_CheckedAppend(stOutputValue, stVariableValue, bInit, (flags AND VisuElems.Visu_InputFlags.Password) = 1, '5');, VisuElemId=-1
    hotkey HotkeyInput Id=481137000448, Key=KeyDown=True, KeyName=NUM6, ActionToExecute=Action=STSnippet=VisuDlg_CheckedAppend(stOutputValue, stVariableValue, bInit, (flags AND VisuElems.Visu_InputFlags.Password) = 1, '6');, VisuElemId=-1
    hotkey HotkeyInput Id=481138049024, Key=KeyDown=True, KeyName=NUM7, ActionToExecute=Action=STSnippet=VisuDlg_CheckedAppend(stOutputValue, stVariableValue, bInit, (flags AND VisuElems.Visu_InputFlags.Password) = 1, '7');, VisuElemId=-1
    hotkey HotkeyInput Id=481139097600, Key=KeyDown=True, KeyName=NUM8, ActionToExecute=Action=STSnippet=VisuDlg_CheckedAppend(stOutputValue, stVariableValue, bInit, (flags AND VisuElems.Visu_InputFlags.Password) = 1, '8');, VisuElemId=-1
    hotkey HotkeyInput Id=481140146176, Key=KeyDown=True, KeyName=NUM9, ActionToExecute=Action=STSnippet=VisuDlg_CheckedAppend(stOutputValue, stVariableValue, bInit, (flags AND VisuElems.Visu_InputFlags.Password) = 1, '9');, VisuElemId=-1
    hotkey HotkeyInput Id=481141194752, Key=KeyDown=True, KeyName=NUM0, ActionToExecute=Action=STSnippet=VisuDlg_CheckedAppend(stOutputValue, stVariableValue, bInit, (flags AND VisuElems.Visu_InputFlags.Password) = 1, '0');, VisuElemId=-1
END_VISUALIZATION

(* stored: Version 1.1.0.1, ProductVersion 3.1.4024.3
   Visu Keypad: Id {6a3e9dc9-120c-41f5-bcf4-244ad38cfac1} *)
